{attribute 'qualified_only'}
VAR_GLOBAL
	//Input
	bStart : BOOL;
	bStop : BOOL;
	bLimitLeft : BOOL;
	bLimitRight : BOOL;
	
	//Output
	bMotorLeft : BOOL;
	bMotorRight : BOOL;
END_VAR

(* stored: Version 1.1.0.1, ProductVersion 3.1.4024.12
   GVL GVL: Id {153a8a10-247c-4ad7-bc40-fd42c82f98bb} *)
